PROGRAM GL11_Transfer
VAR
	GL11: sTransfer;
	GL3: sConveyor;
	GL7: sConveyor;
	GL9: sConveyor;
	GL12: sConveyor;
	GL1_RD: SRoll_Door;
	GL11_PASSSED_ROLL_DOOR : BOOL;
	RUN_FWD_TO_GL3_BIT : BOOL; // GL11 OCCUPIED, GL3 REQUESTING PART, RUN TO GL3 POSITION
	RUN_REV_TO_GL11_BIT : BOOL; //GL11 EMPTY, GL7 OR GL8 REQUESTING PICK UP
	CASE_STOP_UP_REQUEST : BOOL;
END_VAR

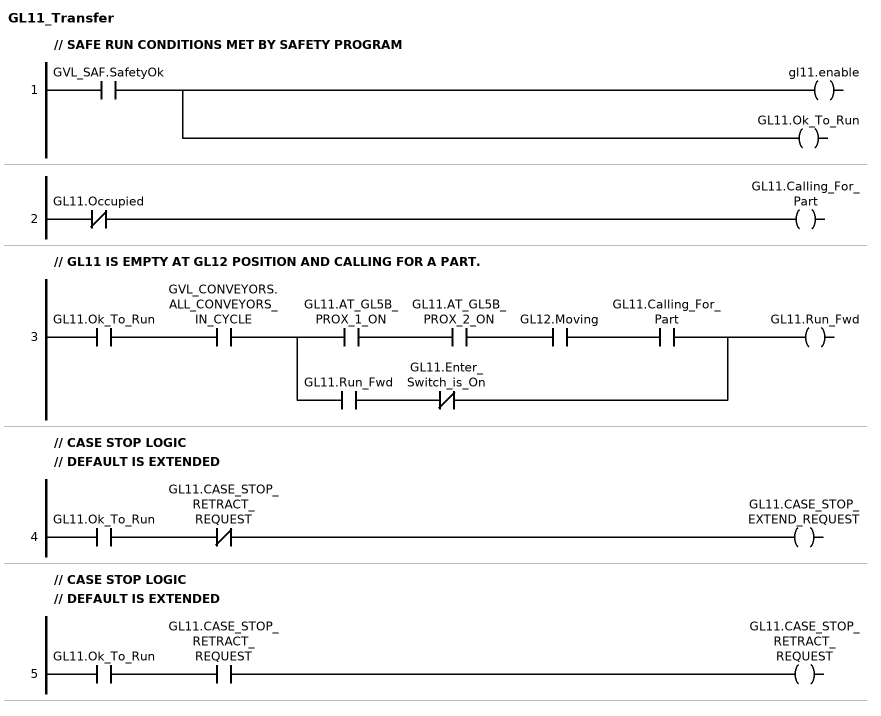
// NETWORK 1: // SAFE RUN CONDITIONS MET BY SAFETY PROGRAM
gl11.enable := GVL_SAF.SafetyOk;
GL11.Ok_To_Run := GVL_SAF.SafetyOk;

// NETWORK 2
GL11.Calling_For_Part := NOT GL11.Occupied;

// NETWORK 3: // GL11 IS EMPTY AT GL12 POSITION AND CALLING FOR A PART.
GL11.Run_Fwd := GL11.Ok_To_Run AND GVL_CONVEYORS.ALL_CONVEYORS_IN_CYCLE AND (GL11.AT_GL5B_PROX_1_ON AND GL11.AT_GL5B_PROX_2_ON AND GL12.Moving AND GL11.Calling_For_Part OR GL11.Run_Fwd AND NOT GL11.Enter_Switch_is_On);

// NETWORK 4: // CASE STOP LOGIC // DEFAULT IS EXTENDED
GL11.CASE_STOP_EXTEND_REQUEST := GL11.Ok_To_Run AND NOT GL11.CASE_STOP_RETRACT_REQUEST;

// NETWORK 5: // CASE STOP LOGIC // DEFAULT IS EXTENDED
GL11.CASE_STOP_RETRACT_REQUEST := GL11.Ok_To_Run AND GL11.CASE_STOP_RETRACT_REQUEST;

END_PROGRAM

(* stored: Version 1.1.0.1, ProductVersion 3.1.4024.12
   POU GL11_Transfer: Id {e34844d7-b1e4-400d-b82f-5a67baafa9a5}, SpecialFunc None *)
